INTERFACE I_PackML_SuspendingCommands

METHOD PUBLIC Abort
VAR_INPUT
END_VAR
END_METHOD

METHOD StateComplete
VAR_INPUT
END_VAR
END_METHOD

METHOD PUBLIC Stop
VAR_INPUT
END_VAR
END_METHOD

END_INTERFACE

(* stored: Version 1.1.0.1, ProductVersion 3.1.4024.12
   Itf I_PackML_SuspendingCommands: Id {293f49ed-8bfe-09e2-1376-339448adb778}
   Method Abort: Id {f5c096e3-e644-0f74-2819-77548df0304c}
   Method StateComplete: Id {b2913adb-125b-063e-33fe-d8bc9b9c9e75}
   Method Stop: Id {78047573-0f7e-0173-10c3-10da67b2aa31} *)
